FUNCTION_BLOCK fb_StnCylinderInOutCtrl
VAR_INPUT
	bEn 								: BOOL;
	bStart			 				: BOOL;
	bCylinderBasketRS_Front			: BOOL;
	bCylinderBasketRS_Back			: BOOL;
	bDeactivatedMode 				: BOOL;
	iCylinderBasketBackDelayTimeSV	: INT;
	iCylinderBasketFrontDelayTimeSV	: INT;

END_VAR
VAR_OUTPUT
	bCylinderBasketAV_Front		: BOOL;
	bCylinderBasketAV_Back		: BOOL;

END_VAR
VAR

	bStep1: BOOL;
	bStep2: BOOL;
	tCylinderBasketBackDelay: TON;
	tCylinderBasketFrontDelay: TON;
END_VAR

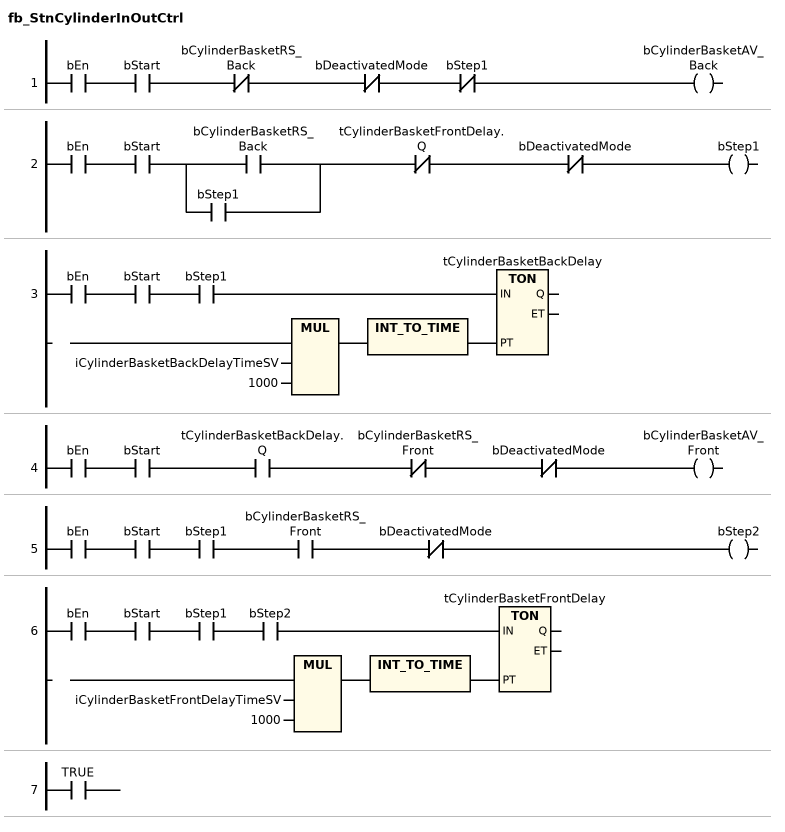
// NETWORK 1
bCylinderBasketAV_Back := bEn AND bStart AND NOT bCylinderBasketRS_Back AND NOT bDeactivatedMode AND NOT bStep1;

// NETWORK 2
bStep1 := (bEn AND bStart AND (bCylinderBasketRS_Back OR bStep1)) AND NOT tCylinderBasketFrontDelay.Q AND NOT bDeactivatedMode;

// NETWORK 3
tCylinderBasketBackDelay(IN := bEn AND bStart AND bStep1, PT := INT_TO_TIME(iCylinderBasketBackDelayTimeSV * 1000)); // TON

// NETWORK 4
bCylinderBasketAV_Front := bEn AND bStart AND tCylinderBasketBackDelay.Q AND NOT bCylinderBasketRS_Front AND NOT bDeactivatedMode;

// NETWORK 5
bStep2 := bEn AND bStart AND bStep1 AND bCylinderBasketRS_Front AND NOT bDeactivatedMode;

// NETWORK 6
tCylinderBasketFrontDelay(IN := bEn AND bStart AND bStep1 AND bStep2, PT := INT_TO_TIME(iCylinderBasketFrontDelayTimeSV * 1000)); // TON

// NETWORK 7

END_FUNCTION_BLOCK

(* stored: Version 1.1.0.1, ProductVersion 3.1.4024.12
   POU fb_StnCylinderInOutCtrl: Id {117bb072-47c4-4372-a491-36ecf9a1934d}, SpecialFunc None *)
